Universal Robots PolyScope program: gravityFeederV.urp

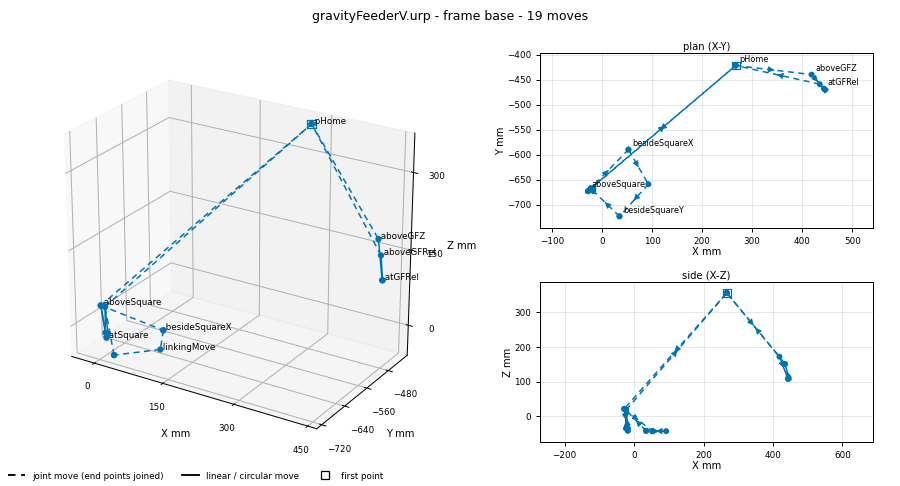
[picture p0: tool path of gravityFeederV.urp in frame base, 19 of 21 moves have a stored position in this frame; points joined in program order, loops and branches not executed]
Program gravityFeederV (installation=admin directory=/programs/THU_530PM/Final createdIn=3.8.0.61336 lastSavedIn=3.15.8.106339 robotSerialNumber=2015350924)
Calibrated DH parameters: a=[0, -0.425, -0.39225, 0, 0, 0]; d=[0.089159, 0, 0, 0.10915, 0.09465, 0.0823]; alpha=[1.570796, 0, 0, 1.570796, -1.570796, 0]; deltaTheta=[0, 0, 0, 0, 0, 0]
Robot Program (runOnlyOnce=true)
  Set DigitalOutput pin=digital_out[0]; digitalValue=0
  Call _adminLinearIndex2
  MoveJ speed 180 deg/s, acceleration 100 deg/s^2 (useActiveTCP=true)
    Waypoint pHome: TCP in base x=267.118 y=-421.457 z=355.823 mm, rx=1.114 ry=1.1062 rz=0.0051 rad; joints [-44.998, -90.002, -90.001, -90.005, 90.001, 0.003] deg; flange x=267.125 y=-421.465 z=431.823 mm, rx=1.2022 ry=-2.9024 rz=-0.0002 rad
    Waypoint aboveGFZ: TCP in base x=418.865 y=-439.595 z=172.117 mm, rx=0.8753 ry=0.8576 rz=-0.0126 rad; joints [-34.991, -106.458, -105.393, -38.795, 86.091, 10.367] deg; flange x=401.249 y=-420.94 z=243.655 mm, rx=-1.1149 ry=2.7612 rz=-0.4823 rad
  MoveL speed 150 mm/s, acceleration 50 mm/s^2 (useActiveTCP=true) feature=Base
    Waypoint atGFRel: TCP in base x=443.443 y=-467.486 z=107.996 mm, rx=0.8755 ry=0.8578 rz=-0.0124 rad; joints [-35.858, -115.926, -102.877, -31.801, 86.386, 9.539] deg; flange x=425.834 y=-448.849 z=179.54 mm, rx=-1.1152 ry=2.7612 rz=-0.4819 rad
    Set DigitalOutput pin=digital_out[0]; digitalValue=1
    Wait Sleep waitTime=1
    Waypoint moveUpRel: TCP in base x=445.78 y=-469.81 z=109.207 mm, rx=0.8754 ry=0.8578 rz=-0.0125 rad; joints [-35.907, -116.184, -102.238, -32.178, 86.396, 9.492] deg; flange x=428.174 y=-451.165 z=180.75 mm, rx=-1.1152 ry=2.7613 rz=-0.482 rad
    Waypoint aboveGFRel: TCP in base x=435.114 y=-458.759 z=151.216 mm, rx=0.8755 ry=0.8579 rz=-0.0125 rad; joints [-35.636, -111.025, -102.567, -37.034, 86.31, 9.748] deg; flange x=417.515 y=-440.125 z=222.764 mm, rx=-1.1153 ry=2.7614 rz=-0.4818 rad
  MoveJ speed 180 deg/s, acceleration 100 deg/s^2 (useActiveTCP=true)
    Waypoint pHome: motionParameters(blendRadius=0.1); TCP in base x=267.118 y=-421.457 z=355.823 mm, rx=1.114 ry=1.1062 rz=0.0051 rad; joints [-44.998, -90.002, -90.001, -90.005, 90.001, 0.003] deg; flange x=267.125 y=-421.465 z=431.823 mm, rx=1.2022 ry=-2.9024 rz=-0.0002 rad
    Waypoint aboveSquare: TCP in base x=-28.511 y=-672.755 z=21.747 mm, rx=1.7065 ry=-0.0121 rz=-1.2064 rad; joints [-83.109, -128.084, -90.371, -51.361, 90.044, 52.13] deg; flange x=-28.598 y=-672.52 z=97.746 mm, rx=1.2074 ry=2.8979 rz=-0.0038 rad
  MoveL speed 250 mm/s, acceleration 1200 mm/s^2 (useActiveTCP=true) feature=Base
    Waypoint atSquare: TCP in base x=-17.891 y=-672.482 z=-41.427 mm, rx=1.7064 ry=-0.0124 rz=-1.2064 rad; joints [-82.196, -133.717, -91.786, -44.3, 90.041, 53.051] deg; flange x=-17.98 y=-672.231 z=34.573 mm, rx=1.2076 ry=2.8977 rz=-0.0041 rad
    Set DigitalOutput pin=digital_out[0]; digitalValue=0
    Wait Sleep waitTime=0.5
    Waypoint aboveSquare: TCP in base x=-28.511 y=-672.755 z=21.747 mm, rx=1.7065 ry=-0.0121 rz=-1.2064 rad; joints [-83.109, -128.084, -90.371, -51.361, 90.044, 52.13] deg; flange x=-28.598 y=-672.52 z=97.746 mm, rx=1.2074 ry=2.8979 rz=-0.0038 rad
    Set DigitalOutput pin=digital_out[0]; digitalValue=1
  MoveJ speed 60 deg/s, acceleration 80 deg/s^2 (useActiveTCP=true)
    Waypoint besideSquareX: TCP in base x=52.617 y=-589.571 z=-42.423 mm, rx=1.7065 ry=-0.0117 rz=-1.2076 rad; joints [-74.267, -126.531, -106.897, -36.426, 89.974, 61.001] deg; flange x=52.598 y=-589.375 z=33.577 mm, rx=1.2085 ry=2.8985 rz=-0.0036 rad
  MoveL speed 35 mm/s, acceleration 35 mm/s^2 (useActiveTCP=true) feature=Base
    If force()≤40 (checkContinuously=true)
      Waypoint atSquareX (Relative): relativeFromPosition TCP in base x=50.865 y=-591.008 z=-41.515 mm, rx=1.7022 ry=-0.008 rz=-1.2089 rad; joints [-74.266, -126.532, -106.898, -36.426, 89.971, 60.977] deg; TCP in base x=-28.314 y=-672.475 z=-41.562 mm, rx=1.7067 ry=-0.0121 rz=-1.2064 rad; joints [-83.089, -133.766, -91.707, -44.351, 90.046, 52.151] deg; flange x=-28.404 y=-672.249 z=34.438 mm, rx=1.2075 ry=2.8979 rz=-0.0036 rad
    Wait Sleep waitTime=0.5
  MoveJ speed 60 deg/s, acceleration 80 deg/s^2 (useActiveTCP=true)
    Waypoint besideSquareX: TCP in base x=52.617 y=-589.571 z=-42.423 mm, rx=1.7065 ry=-0.0117 rz=-1.2076 rad; joints [-74.267, -126.531, -106.897, -36.426, 89.974, 61.001] deg; flange x=52.598 y=-589.375 z=33.577 mm, rx=1.2085 ry=2.8985 rz=-0.0036 rad
    Waypoint linkingMove: motionParameters(blendRadius=0.01); TCP in base x=92.406 y=-658.703 z=-42.29 mm, rx=1.7071 ry=-0.0114 rz=-1.2067 rad; joints [-72.572, -133.085, -93.255, -43.522, 90.01, 62.663] deg; flange x=92.339 y=-658.532 z=33.709 mm, rx=1.2075 ry=2.8984 rz=-0.0027 rad
    Waypoint besideSquareY: TCP in base x=34.628 y=-723.042 z=-41.53 mm, rx=1.7068 ry=-0.0118 rz=-1.2057 rad; joints [-78.597, -138.866, -81.159, -49.796, 90.051, 56.613] deg; flange x=34.515 y=-722.822 z=34.47 mm, rx=1.2066 ry=2.8979 rz=-0.0033 rad
  MoveL speed 35 mm/s, acceleration 35 mm/s^2 (useActiveTCP=true) feature=Base
    If force()≤40 (checkContinuously=true)
      Waypoint atSquareY (Relative): relativeFromPosition TCP in base x=32.384 y=-724.404 z=-40.504 mm, rx=1.7021 ry=-0.0085 rz=-1.209 rad; joints [-78.599, -138.865, -81.161, -49.795, 90.053, 56.612] deg; TCP in base x=-15.805 y=-673.754 z=-41.467 mm, rx=1.7062 ry=-0.0122 rz=-1.2065 rad; joints [-82.03, -133.837, -91.546, -44.419, 90.028, 53.212] deg; flange x=-15.879 y=-673.5 z=34.533 mm, rx=1.2075 ry=2.8979 rz=-0.0043 rad
    Wait Sleep waitTime=0.5
  MoveJ speed 60 deg/s, acceleration 80 deg/s^2 (useActiveTCP=true)
    Waypoint besideSquareY: TCP in base x=34.628 y=-723.042 z=-41.53 mm, rx=1.7068 ry=-0.0118 rz=-1.2057 rad; joints [-78.597, -138.866, -81.159, -49.796, 90.051, 56.613] deg; flange x=34.515 y=-722.822 z=34.47 mm, rx=1.2066 ry=2.8979 rz=-0.0033 rad
    Waypoint aboveSquareNew: TCP in base x=-22.971 y=-667.274 z=18.45 mm, rx=1.7065 ry=-0.0121 rz=-1.2064 rad; joints [-82.573, -127.757, -91.596, -50.461, 90.041, 52.664] deg; flange x=-23.057 y=-667.037 z=94.449 mm, rx=1.2074 ry=2.8979 rz=-0.0038 rad
    Set DigitalOutput pin=digital_out[0]; digitalValue=0
    Wait Sleep waitTime=1
  MoveL speed 250 mm/s, acceleration 1200 mm/s^2 (useActiveTCP=true) feature=Base
    Waypoint atSquareNew: TCP in base x=-23.327 y=-667.602 z=-34.524 mm, rx=1.7078 ry=-0.0434 rz=-1.2108 rad; joints [-82.736, -132.559, -92.965, -43.61, 90.578, 53.735] deg; flange x=-24.233 y=-666.559 z=41.464 mm, rx=1.2328 ry=2.8718 rz=-0.0123 rad
    Set DigitalOutput pin=digital_out[0]; digitalValue=1
    Wait Sleep waitTime=1
    Waypoint easeout: TCP in base x=-17.567 y=-667.635 z=-34.572 mm, rx=1.7078 ry=-0.0434 rz=-1.2109 rad; joints [-82.238, -132.549, -92.995, -43.588, 90.569, 54.238] deg; flange x=-18.471 y=-666.597 z=41.415 mm, rx=1.233 ry=2.8718 rz=-0.0123 rad
    Waypoint aboveSquareNew: TCP in base x=-22.971 y=-667.274 z=18.45 mm, rx=1.7065 ry=-0.0121 rz=-1.2064 rad; joints [-82.573, -127.757, -91.596, -50.461, 90.041, 52.664] deg; flange x=-23.057 y=-667.037 z=94.449 mm, rx=1.2074 ry=2.8979 rz=-0.0038 rad
  MoveJ speed 60 deg/s, acceleration 80 deg/s^2 (useActiveTCP=true)
    Waypoint pHome: TCP in base x=267.118 y=-421.457 z=355.823 mm, rx=1.114 ry=1.1062 rz=0.0051 rad; joints [-44.998, -90.002, -90.001, -90.005, 90.001, 0.003] deg; flange x=267.125 y=-421.465 z=431.823 mm, rx=1.2022 ry=-2.9024 rz=-0.0002 rad
SubProgram  [hidden by the author, left out]
SubProgram _adminLinearIndex2 [hidden by the author, left out]
